PROGRAM z_CONTROL
VAR
	{attribute 'old_input_assignments' := ''}
	PULSO: PULS_1S;
END_VAR

PULSO(Q=> );
(*-------------------------------------------------------------------------------------------------------*)
(*P402 Piloto Cala Alarma*)


(*-------------------------------------------------------------------------------------------------------*)
(*P405 Sirena Alarma*)



(*-------------------------------------------------------------------------------------------------------*)
(*P403 Piloto Continua Programa*)

END_PROGRAM

(* stored: Version 1.1.0.1, ProductVersion 3.1.4024.10
   POU z_CONTROL: Id {2da1a52e-dc32-49c2-8b8d-e3c17fe3e629}, SpecialFunc None *)
